INTERFACE I_Context EXTENDS I_Object

END_INTERFACE

(* stored: Version 1.1.0.1, ProductVersion 3.1.4024.12
   Itf I_Context: Id {b6c47ed1-8af3-469c-b461-117a3f997fa8} *)
